ABB RobotStudio station: FinalProject_SP.rspag

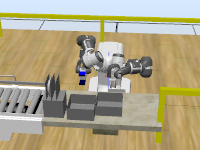
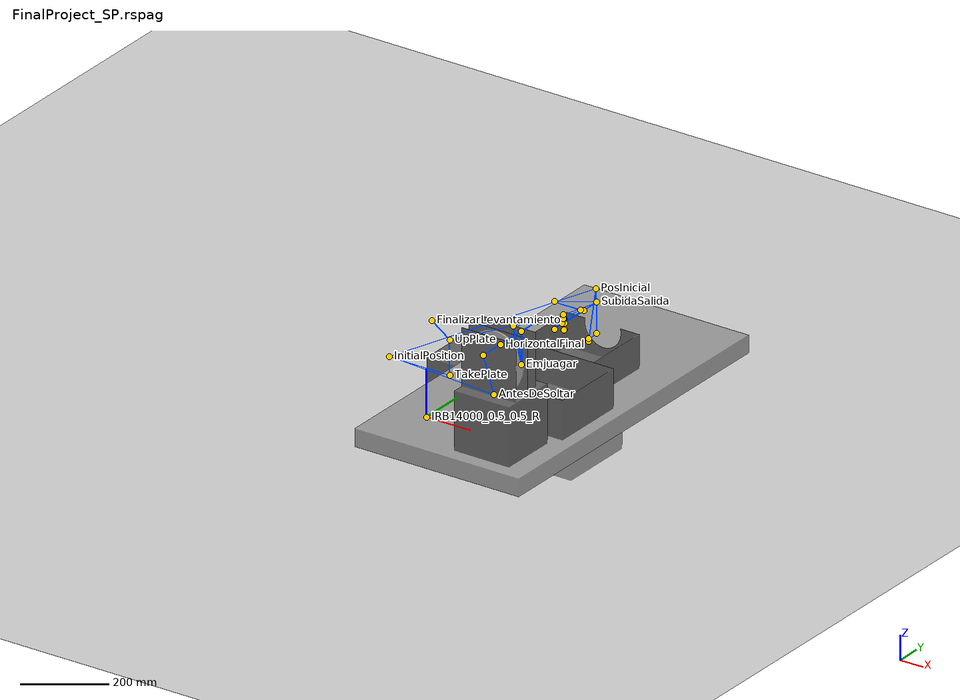
[picture v1: parts stored in the station drawn from their meshes, with robot base, taught points and paths (robot models come from the ABB library and are not in the file)]
--- station ---
Station FinalProject_SP (saved by RobotStudio 21.3.9648.0)
Controller IRB14000_1
  mechanical unit ROB_R: IRB14000_0.5_0.5_R, 6 joints, base frame (0, 0, 0) mm
  mechanical unit ROB_R_7: IRB14000_0.5_0.5_R, 1 joints, base frame (0, 0, 0) mm
  mechanical unit ROB_L: IRB14000_0.5_0.5_L, 6 joints, base frame (0, 0, 0) mm
  mechanical unit ROB_L_7: IRB14000_0.5_0.5_L, 1 joints, base frame (0, 0, 0) mm
Layout (positions relative to the parent item):
  - IRB14000_0.5_0.5 [mechanism, from Robots\IRB14000_0.5_0.5__01.rslib] at (0, 0, 0) mm
  - IRB14000_0.5_0.5_R [mechanism, from Robots\IRB14000_0.5_0.5__01.rslib] at (0, 0, 0) mm; joint values [-0.1923, -2.1323, -2.3764, 0.5232, 0.2776, 1.3361, 0.0448] (rad or m)
  - IRB14000_0.5_0.5_L [mechanism, from Robots\IRB14000_0.5_0.5__01.rslib] at (0, 0, 0) mm; joint values [2.2057, 0.7592, -2.9409, 0.6294, 1.2654, 1.781, -1.09] (rad or m)
  - LeftTool [mechanism] at (420.61, 55.54, 501.86) mm, rotated rx 176.45 ry 0.33 rz 178.52 deg; joint values [0, 0] (rad or m)
      TCP LeftTool_1 at (0, 0, 87) mm
      links: MainBody, R_Wash, L_Dry
  - floor [part] at (-1635.16, -1487.82, 4.97) mm, size 3000 x 3000 x 1 mm
  - Table [part] at (136.38, -477.32, 155.93) mm, size 450 x 900 x 45 mm
  - Plate [part] at (464.91, -410.88, 426.41) mm, rotated rx -91 ry -6 rz 0 deg, size 150 x 150 x 20 mm
  - SinkWsoap_3 [part] at (290.47, -67.3, 205.89) mm, size 200 x 200 x 85 mm
  - Sink_2 [part] at (461.13, -169.65, 206.31) mm, size 200 x 200 x 100 mm
  - Pieza_5 [part] at (260.22, -92.11, 0) mm, size 200 x 200 x 160 mm
  - RightGrip [mechanism] at (-31.94, -222.15, 256.56) mm, rotated rx -153.04 ry -89.35 rz -27.45 deg; joint values [0] (rad or m)
      TCP RightGrip at (0, 0, 85) mm
      links: Base, RightFinger, LeftFinger
  - 400_guide_2 [part, from Equipment\Conveyor Guide 400.rslib] at (524.45, -3451.19, -560.07) mm, rotated rx 0 ry 0 rz 89.33 deg
  - Pieza_8 [part] at (382.54, -381.93, 349.62) mm, size 159 x 2 x 150 mm
  - Pieza_9 [part] at (387.36, -418.51, 350.42) mm, size 150 x 1 x 150 mm
  - Pieza_10 [part] at (388.58, -447.06, 203.31) mm, size 150 x 150 x 150 mm
  - Pieza_11 [part], size 150 x 150 x 150 mm
  - Pieza_12 [part] at (388.74, -344.82, 350.01) mm, size 150 x 2 x 150 mm
  - Fence_2500_2 [graphiccomponentgroup, from Equipment\Fence_2500.rslib] at (-957.65, -1356.65, -1537.2) mm
    - Body 1 [part, from Equipment\Fence_2500.rslib]
    - Body 2 [part, from Equipment\Fence_2500.rslib]
  - Gate_2 [graphiccomponentgroup, from Equipment\Fence_Gate.rslib] at (-1379.63, -1420.32, -1615.31) mm, rotated rx 0 ry 0 rz -88.3 deg
    - Body 1 [part, from Equipment\Fence_Gate.rslib]
    - Body 2 [part, from Equipment\Fence_Gate.rslib]
    - Body 3 [part, from Equipment\Fence_Gate.rslib]
  - Gate_3 [graphiccomponentgroup, from Equipment\Fence_Gate.rslib] at (522.14, 1119.74, -1537.29) mm, rotated rx 0 ry 0 rz 90.8 deg
    - Body 1 [part, from Equipment\Fence_Gate.rslib]
    - Body 2 [part, from Equipment\Fence_Gate.rslib]
    - Body 3 [part, from Equipment\Fence_Gate.rslib]
  - Fence_740_2 [graphiccomponentgroup, from Equipment\Fence_740.rslib] at (506.71, 414.21, -1523.62) mm
    - Body 1 [part, from Equipment\Fence_740.rslib]
    - Body 2 [part, from Equipment\Fence_740.rslib]
Attachment: LeftTool is attached to IRB14000_0.5_0.5_L / Link7
Attachment: RightGrip is attached to IRB14000_0.5_0.5_R / Link7
EventTableEntry 3566: Group=, Trigger=DO_CloseGrip 3567, Actions=[EventTableActionMechanicalPose 3568, EventTableActionAttach 3576], Comment=, ActivationMode=2, Cyclic=false
EventTableTriggerIO 3567: IOValue=[1], IRC5Controller=? -1, Operator=0, SignalSource=IRB14000_1 1167
EventTableActionMechanicalPose 3568: VirtualSignal=SS_GripperClosed, Mechanism=RightGrip 3516, ToPoseName=Cerrado, VirtualSignalValue=[1]
EventTableEntry 3569: Group=, Trigger=DO_CloseGrip 3570, Actions=[EventTableActionMechanicalPose 5234, EventTableActionDetach 5235], Comment=, ActivationMode=2, Cyclic=false
EventTableTriggerIO 3570: IOValue=[0], IRC5Controller=? -1, Operator=0, SignalSource=IRB14000_1 1167
EventTableEntry 3572: Group=, Trigger=NOP 3573, Actions=[DI_GripperClosed 3575], Comment=, ActivationMode=2, Cyclic=false
EventTableTriggerLogic 3573: layoutX=8, layoutY=16, Operand1=SS_GripperClosed 3574, Operand2=? -1, Operator=4, Delay=1000
EventTableTriggerIO 3574: IOValue=[-1], IRC5Controller=? -1, Operator=0, SignalSource=FinalProject_SP 1
EventTableActionIO 3575: IOValue=[-1], IRC5Controller=? -1, SignalTarget=IRB14000_1 1167
EventTableActionAttach 3576: AttachmentParent=RightGrip 3516, AttachmentChild=Plate 3480, MountObject=false, Offset=[X=1, Y=0, Z=0, W=0, X=0, Y=1, Z=0, W=0, X=0, Y=0, Z=1, W=0, X=0, Y=0, Z=0, W=1], FlangeIndext=0, FindNearest=false
EventTableActionMechanicalPose 5234: VirtualSignal=SS_GripperClosed, Mechanism=RightGrip 3516, ToPoseName=Abierto, VirtualSignalValue=[0]
EventTableActionDetach 5235: AttachmentParent=RightGrip 3516, AttachmentChild=Plate 3480
EventTableTriggerIO 5306: IOValue=[1], IRC5Controller=? -1, Operator=0, SignalSource=IRB14000_1 1167
EventTableTriggerIO 5307: IOValue=[1], IRC5Controller=? -1, Operator=0, SignalSource=IRB14000_1 1167
EventTableTriggerIO 5308: IOValue=[0], IRC5Controller=? -1, Operator=0, SignalSource=IRB14000_1 1167
EventTableTriggerIO 5309: IOValue=[0], IRC5Controller=? -1, Operator=0, SignalSource=IRB14000_1 1167
EventTableTriggerLogic 5310: layoutX=8, layoutY=16, Operand1=SS_GripperClosed 3574, Operand2=? -1, Operator=4, Delay=1000
EventTableTriggerLogic 5311: layoutX=8, layoutY=16, Operand1=SS_GripperClosed 3574, Operand2=? -1, Operator=4, Delay=1000
Station signals: DI SS_GripperClosed
Targets, tools, work objects and paths stored in the station and not in the controller backup, written as RAPID:
! task T_ROB_R
MODULE Module1
  CONST robtarget SoltarObjeto:=[[612.086300085,-497.889224852,286.694545259],[0.048207182,0.789967534,-0.030176126,0.610505335],[1,1,1,4],[88.920010699,9E+09,9E+09,9E+09,9E+09,9E+09]];
ENDMODULE


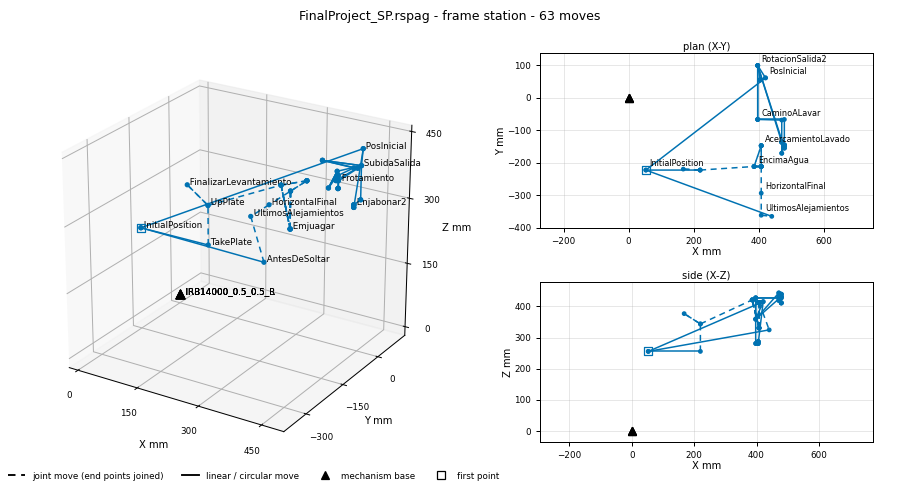
[picture p0: tool path of FinalProject_SP.rspag in frame station, 63 of 63 moves have a stored position in this frame; points joined in program order, loops and branches not executed]
--- Backups/IRB14000_1/RAPID/TASK1/PROGMOD/CalibData.mod ---
MODULE CalibData
    PERS tooldata RightGrip:=[TRUE,[[0,0,85],[1,0,0,0]],[0.32367,[0,0,17.36],[1,0,0,0],0,0,0]];
ENDMODULE

--- Backups/IRB14000_1/RAPID/TASK1/PROGMOD/Module1.mod ---
MODULE Module1
        CONST robtarget InitialPosition:=[[53.055314104,-222.870016919,255.704154577],[0.001177788,0.710631418,-0.004820161,0.703546989],[0,0,0,4],[-96.630018739,9E+09,9E+09,9E+09,9E+09,9E+09]];
    CONST robtarget TakePlate:=[[220.05553838,-222.870371261,255.704183843],[0.001177763,0.71063163,-0.004819912,0.703546777],[0,0,0,4],[-96.630024002,9E+09,9E+09,9E+09,9E+09,9E+09]];
    CONST robtarget UpPlate:=[[220.056150571,-222.871159309,343.704161267],[0.001177802,0.710632144,-0.004819416,0.703546262],[0,0,0,4],[-96.63002197,9E+09,9E+09,9E+09,9E+09,9E+09]];
    CONST robtarget FinalizarLevantamiento:=[[168.058261278,-219.873083697,376.704096677],[0.507683817,0.497248487,0.498428155,0.496558615],[0,1,-1,4],[-156.301628385,9E+09,9E+09,9E+09,9E+09,9E+09]];
    CONST robtarget Rotacion:=[[220.057272902,-222.872151334,343.70419509],[0.507684048,0.497248575,0.498427407,0.496559041],[0,0,-1,4],[-96.630018769,9E+09,9E+09,9E+09,9E+09,9E+09]];
    CONST robtarget EncimaAgua:=[[386.063679666,-211.876833518,420.702145472],[0.328812168,0.626355418,0.630919785,0.318593273],[0,2,-1,4],[98.779984801,9E+09,9E+09,9E+09,9E+09,9E+09]];
    CONST robtarget Emjuagar:=[[408.064481901,-211.877451805,330.701831056],[0.284000479,0.64705336,0.65232018,0.274124169],[0,2,-1,4],[102.139980128,9E+09,9E+09,9E+09,9E+09,9E+09]];
    CONST robtarget SalirDelAgua:=[[408.065294918,-211.877887738,412.70165188],[0.533074265,0.470579483,0.471179643,0.521897042],[-1,2,-1,4],[102.139982595,9E+09,9E+09,9E+09,9E+09,9E+09]];
    CONST robtarget AcomodoParaLavar:=[[408.065461711,-147.878021494,412.701612854],[0.53307426,0.470579475,0.471179771,0.521896939],[-1,2,-1,4],[102.139981571,9E+09,9E+09,9E+09,9E+09,9E+09]];
    CONST robtarget AcercamientoLavado:=[[408.066683421,-147.878727164,412.701031749],[0.533073873,0.470579276,0.471180857,0.521896533],[-1,2,-1,4],[102.139981352,9E+09,9E+09,9E+09,9E+09,9E+09]];
    CONST robtarget acercamiento2Lavado:=[[408.067566131,-147.879323271,412.700510834],[0.688610388,0.177278397,0.656761973,0.251101203],[0,2,-2,4],[122.539973578,9E+09,9E+09,9E+09,9E+09,9E+09]];
    CONST robtarget acercamiento2Lavado_2:=[[408.067566131,-147.879323271,412.700510834],[0.688610388,0.177278397,0.656761973,0.251101203],[0,2,-2,4],[122.539973578,9E+09,9E+09,9E+09,9E+09,9E+09]];
    CONST robtarget Emjuagar_2:=[[408.064481901,-211.877451805,330.701831056],[0.284000479,0.64705336,0.65232018,0.274124169],[0,2,-1,4],[102.139980128,9E+09,9E+09,9E+09,9E+09,9E+09]];
    CONST robtarget SalirDelAgua_2:=[[408.065294918,-211.877887738,412.70165188],[0.533074265,0.470579483,0.471179643,0.521897042],[-1,2,-1,4],[102.139982595,9E+09,9E+09,9E+09,9E+09,9E+09]];
    CONST robtarget Emjuagar_2_2:=[[408.064481901,-211.877451805,330.701831056],[0.284000479,0.64705336,0.65232018,0.274124169],[0,2,-1,4],[102.139980128,9E+09,9E+09,9E+09,9E+09,9E+09]];
    CONST robtarget SalirDelAgua_2_2:=[[408.065294918,-211.877887738,412.70165188],[0.533074265,0.470579483,0.471179643,0.521897042],[-1,2,-1,4],[102.139982595,9E+09,9E+09,9E+09,9E+09,9E+09]];
    CONST robtarget UltimoAlejamiento:=[[408.07197068,-293.881092513,412.699267968],[0.533045558,0.470580996,0.471214617,0.521893422],[-1,1,-1,4],[88.459990285,9E+09,9E+09,9E+09,9E+09,9E+09]];
    CONST robtarget HorizontalFinal:=[[408.072778957,-293.881627629,412.69925656],[0.044169035,0.709671302,-0.035834669,0.702233306],[-1,2,0,4],[80.980024532,9E+09,9E+09,9E+09,9E+09,9E+09]];
    CONST robtarget DejaElPlato:=[[408.076946424,-361.884549979,286.698372064],[0.044168859,0.709673429,-0.035831454,0.702231331],[-2,2,0,4],[94.167708654,9E+09,9E+09,9E+09,9E+09,9E+09]];
    CONST robtarget UltimosAlejamientos:=[[408.072401892,-361.881327349,412.699273877],[0.533045426,0.470580989,0.471214987,0.521893229],[-1,1,-1,4],[88.45998457,9E+09,9E+09,9E+09,9E+09,9E+09]];
    CONST robtarget AntesDeSoltar:=[[440.491875375,-365.351645888,324.606650036],[0.020610194,-0.811420808,-0.004875566,-0.584078523],[-1,1,0,4],[88.499974458,9E+09,9E+09,9E+09,9E+09,9E+09]];
!***********************************************************
    !***********************************************************
    PROC main()
        !Añada aquí su código
        MoveL InitialPosition,v500,fine,RightGrip\WObj:=wobj0;
        WaitDI DI_GripperClosed,0; !Gripper is opened
        MoveL TakePlate,v500,fine,RightGrip\WObj:=wobj0;
        SetDO DO_CloseGrip,1; !Close the gripper
        WaitDI DI_GripperClosed,1;!Gripper is closed
        MoveJ UpPlate,v500,z100,RightGrip\WObj:=wobj0;
        MoveJ FinalizarLevantamiento,v500,z100,RightGrip\WObj:=wobj0;
        MoveJ Rotacion,v500,z100,RightGrip\WObj:=wobj0;
        MoveJ EncimaAgua,v500,z100,RightGrip\WObj:=wobj0;
        MoveJ Emjuagar,v500,z100,RightGrip\WObj:=wobj0;
        MoveJ EncimaAgua,v500,z100,RightGrip\WObj:=wobj0;
        MoveJ Emjuagar,v500,z100,RightGrip\WObj:=wobj0;
        MoveJ SalirDelAgua,v500,fine,RightGrip\WObj:=wobj0;
        MoveJ Emjuagar_2,v500,z100,RightGrip\WObj:=wobj0;
        MoveJ SalirDelAgua_2,v500,fine,RightGrip\WObj:=wobj0;
        MoveJ Emjuagar_2_2,v500,z100,RightGrip\WObj:=wobj0;
        MoveJ SalirDelAgua_2_2,v500,fine,RightGrip\WObj:=wobj0;
        MoveJ AcercamientoLavado,v200,fine,RightGrip\WObj:=wobj0;
        MoveJ acercamiento2Lavado,v80,fine\Inpos:=stoptime1_5,RightGrip\WObj:=wobj0;
        MoveJ EncimaAgua,v500,fine,RightGrip\WObj:=wobj0;
        MoveJ Emjuagar,v500,fine,RightGrip\WObj:=wobj0;
        MoveJ EncimaAgua,v500,fine,RightGrip\WObj:=wobj0;
        MoveJ AcercamientoLavado,v500,fine,RightGrip\WObj:=wobj0;
        MoveJ acercamiento2Lavado,v500,fine\Inpos:=stoptime1_5,RightGrip\WObj:=wobj0;
        MoveJ AcercamientoLavado,v500,fine,RightGrip\WObj:=wobj0;
        MoveJ HorizontalFinal,v500,fine,RightGrip\WObj:=wobj0;
        MoveJ UltimosAlejamientos,v500,fine,RightGrip\WObj:=wobj0;
        MoveJ AntesDeSoltar,v1000,z100,RightGrip\WObj:=wobj0;
        WaitDI DI_GripperClosed,1; !Gripper is closed
        SetDO DO_CloseGrip,0; !Open the gripper
        WaitDI DI_GripperClosed,0;!Gripper is Open
        MoveL InitialPosition,v500,fine,RightGrip\WObj:=wobj0;

    ENDPROC
ENDMODULE

--- Backups/IRB14000_1/RAPID/TASK2/PROGMOD/CalibData.mod ---
MODULE CalibData
    PERS tooldata Dryer_Washer_1:=[TRUE,[[0,0,87],[1,0,0,0]],[0.306692,[0,-1.008,28.95],[1,0,0,0],0,0,0]];
    PERS tooldata Servo:=[TRUE,[[0,0,114.2],[1,0,0,0]],[0.229,[7.9,12.4,48.7],[1,0,0,0],0.00021,0.00023,0.00008]];
    PERS tooldata Camera:=[TRUE,[[-7.3,28.3,35.1],[0.5,-0.5,0.5,0.5]],[0.229,[7.9,12.4,48.7],[1,0,0,0],0.00021,0.00023,0.00008]];
    PERS tooldata LeftTool_1:=[TRUE,[[0,0,87],[1,0,0,0]],[0.30618,[0,-1.009,28.951],[1,0,0,0],0,0,0]];
ENDMODULE

--- Backups/IRB14000_1/RAPID/TASK2/PROGMOD/Module1.mod ---
MODULE Module1
        CONST robtarget PosInicial:=[[421.244619941,60.912152429,415.028508411],[0.003235703,0.012822081,0.999433724,0.030941171],[1,1,-1,0],[-178.213591377,9E+09,9E+09,9E+09,9E+09,9E+09]];
    CONST robtarget SegundaPos:=[[531.247516921,296.914105526,415.026910938],[0.003233398,0.012823194,0.999433674,0.030942565],[2,1,0,0],[-152.08998148,9E+09,9E+09,9E+09,9E+09,9E+09]];
    CONST robtarget AcomodoJabon:=[[531.249287785,296.915302981,283.026126749],[0.003677623,0.012703494,0.999904722,-0.003955191],[2,1,0,0],[-152.089982592,9E+09,9E+09,9E+09,9E+09,9E+09]];
    CONST robtarget SegundoAcomodo:=[[531.251888568,200.917989137,287.024191767],[0.003743422,-0.004748162,0.999974161,-0.003888287],[2,1,0,0],[-151.229980314,9E+09,9E+09,9E+09,9E+09,9E+09]];
    CONST robtarget Encaje:=[[531.253237835,180.919326703,287.022987741],[0.000816881,0.005991691,-0.69184437,0.722021329],[1,0,0,0],[-151.230030681,9E+09,9E+09,9E+09,9E+09,9E+09]];
    CONST robtarget Lavar:=[[531.256510861,180.923529425,243.019596759],[0.691724056,0.721807274,0.012895058,-0.018595875],[1,0,2,0],[-151.230032118,9E+09,9E+09,9E+09,9E+09,9E+09]];
    CONST robtarget BajaASoap:=[[421.245417577,58.912937477,271.02790989],[0.003234896,0.012822498,0.999433703,0.030941751],[1,1,-1,0],[-168.160186005,9E+09,9E+09,9E+09,9E+09,9E+09]];
    CONST robtarget Enjabonar:=[[405.248437711,54.917136531,281.025032798],[0.704216771,0.709627455,0.013003664,-0.018398897],[1,0,-1,0],[-152.810020426,9E+09,9E+09,9E+09,9E+09,9E+09]];
    CONST robtarget Enjabonar2:=[[405.249506318,54.918706238,287.024012367],[0.704215896,0.709628284,0.01300405,-0.018400126],[1,0,-1,0],[-152.810017528,9E+09,9E+09,9E+09,9E+09,9E+09]];
    CONST robtarget RotacionSalida:=[[405.250228712,54.919564027,287.023505096],[0.221162905,0.974976545,0.020779228,-0.00871373],[2,1,-3,0],[-151.089999947,9E+09,9E+09,9E+09,9E+09,9E+09]];
    CONST robtarget RotacionSalida2:=[[397.251225339,98.920933427,281.022531986],[0.221162073,0.974976732,0.02077867,-0.008715334],[2,1,-2,0],[-144.406554524,9E+09,9E+09,9E+09,9E+09,9E+09]];
    CONST robtarget SalidaRotacion:=[[397.257647968,98.928500253,325.017724075],[0.047711709,0.997734001,0.026081142,-0.039626132],[2,1,-3,0],[-141.807190023,9E+09,9E+09,9E+09,9E+09,9E+09]];
    CONST robtarget AfueraRotacion:=[[397.252338551,98.922405636,281.021643738],[0.704213985,0.709630106,0.01300311,-0.018403658],[2,0,-1,0],[-143.450011398,9E+09,9E+09,9E+09,9E+09,9E+09]];
    CONST robtarget SubidaSalida:=[[397.253299337,98.923503411,359.020949108],[0.704213348,0.709630696,0.01300383,-0.018404812],[2,0,-1,0],[-137.099990443,9E+09,9E+09,9E+09,9E+09,9E+09]];
    CONST robtarget CaminoALavar:=[[397.254740388,-67.075582852,427.02014683],[0.704212985,0.709631027,0.013003711,-0.018405994],[2,-1,-1,0],[-138.173949069,9E+09,9E+09,9E+09,9E+09,9E+09]];
    CONST robtarget AcercamientoLavado:=[[397.255236135,-67.075179426,427.019791885],[0.465965923,0.88451561,0.017817153,-0.013800111],[2,0,-3,0],[-162.169977355,9E+09,9E+09,9E+09,9E+09,9E+09]];
    CONST robtarget Acercamiento2:=[[479.255350173,-67.075059648,427.019646749],[0.465965804,0.884515669,0.017817213,-0.013800279],[1,0,-2,0],[-162.169971229,9E+09,9E+09,9E+09,9E+09,9E+09]];
    CONST robtarget Frotamiento:=[[479.256631089,-145.074003616,427.018181948],[0.465964987,0.884516076,0.01781704,-0.013802011],[1,0,-3,0],[-162.170033234,9E+09,9E+09,9E+09,9E+09,9E+09]];
    CONST robtarget Bajo1:=[[479.257332601,-145.073375587,411.017323942],[0.465964389,0.88451639,0.017816677,-0.013802499],[1,0,-3,0],[-161.630016937,9E+09,9E+09,9E+09,9E+09,9E+09]];
    CONST robtarget Bajo2:=[[479.257619446,-147.073077759,411.016894097],[0.465964074,0.88451655,0.017816607,-0.013802987],[1,0,-3,0],[-161.630015461,9E+09,9E+09,9E+09,9E+09,9E+09]];
    CONST robtarget RotacionPenultima:=[[479.257920024,-147.072880521,411.016622834],[0.826677125,0.562225014,0.009251006,-0.020551967],[1,-1,-1,0],[-161.339982134,9E+09,9E+09,9E+09,9E+09,9E+09]];
    CONST robtarget CambioDeLado:=[[479.258634617,-147.072192495,411.01554837],[0.00925188,0.020552151,-0.826677374,0.562224626],[1,0,0,0],[-161.339985535,9E+09,9E+09,9E+09,9E+09,9E+09]];
    CONST robtarget Frotamiento2:=[[479.26034828,-147.070681628,439.013141409],[0.009254109,0.020552461,-0.826678168,0.562223411],[1,0,0,0],[-161.339982258,9E+09,9E+09,9E+09,9E+09,9E+09]];
    CONST robtarget BajadaLimpia:=[[479.261993602,-155.069467218,431.011459943],[0.009256027,0.020552551,-0.826678574,0.56222278],[1,0,0,0],[-161.340012683,9E+09,9E+09,9E+09,9E+09,9E+09]];
    CONST robtarget CaminoALavar_2:=[[397.254740388,-67.075582852,427.02014683],[0.704212985,0.709631027,0.013003711,-0.018405994],[2,-1,-1,0],[-138.173949069,9E+09,9E+09,9E+09,9E+09,9E+09]];
    CONST robtarget AcercamientoLavado_2:=[[397.255236135,-67.075179426,427.019791885],[0.465965923,0.88451561,0.017817153,-0.013800111],[2,0,-3,0],[-162.169977355,9E+09,9E+09,9E+09,9E+09,9E+09]];
    CONST robtarget Acercamiento2_2:=[[479.255350173,-67.075059648,427.019646749],[0.465965804,0.884515669,0.017817213,-0.013800279],[1,0,-2,0],[-162.169971229,9E+09,9E+09,9E+09,9E+09,9E+09]];
    CONST robtarget Frotamiento_2:=[[479.256631089,-145.074003616,427.018181948],[0.465964987,0.884516076,0.01781704,-0.013802011],[1,0,-3,0],[-162.170033234,9E+09,9E+09,9E+09,9E+09,9E+09]];
    CONST robtarget Bajo1_2:=[[479.257332601,-145.073375587,411.017323942],[0.465964389,0.88451639,0.017816677,-0.013802499],[1,0,-3,0],[-161.630016937,9E+09,9E+09,9E+09,9E+09,9E+09]];
    CONST robtarget Bajo2_2:=[[479.257619446,-147.073077759,411.016894097],[0.465964074,0.88451655,0.017816607,-0.013802987],[1,0,-3,0],[-161.630015461,9E+09,9E+09,9E+09,9E+09,9E+09]];
    CONST robtarget RotacionPenultima_2:=[[479.257920024,-147.072880521,411.016622834],[0.826677125,0.562225014,0.009251006,-0.020551967],[1,-1,-1,0],[-161.339982134,9E+09,9E+09,9E+09,9E+09,9E+09]];
    CONST robtarget Frotamiento2_2:=[[479.26034828,-147.070681628,439.013141409],[0.009254109,0.020552461,-0.826678168,0.562223411],[1,0,0,0],[-161.339982258,9E+09,9E+09,9E+09,9E+09,9E+09]];
    CONST robtarget BajadaLimpia_3:=[[479.261993602,-155.069467218,431.011459943],[0.009256027,0.020552551,-0.826678574,0.56222278],[1,0,0,0],[-161.340012683,9E+09,9E+09,9E+09,9E+09,9E+09]];
    CONST robtarget BajadaLimpia_2:=[[479.261993602,-155.069467218,431.011459943],[0.009256027,0.020552551,-0.826678574,0.56222278],[1,0,0,0],[-161.340012683,9E+09,9E+09,9E+09,9E+09,9E+09]];
    CONST robtarget Frotamiento2_3:=[[479.26034828,-147.070681628,439.013141409],[0.009254109,0.020552461,-0.826678168,0.562223411],[1,0,0,0],[-161.339982258,9E+09,9E+09,9E+09,9E+09,9E+09]];
    CONST robtarget UltimaAproximacion:=[[471.256137044,-69.074277916,427.018433556],[0.465965108,0.884516007,0.017817773,-0.013801412],[1,0,-2,0],[-161.699970308,9E+09,9E+09,9E+09,9E+09,9E+09]];
    CONST robtarget UltimoToque:=[[471.257048398,-137.073488671,433.016805154],[0.46596401,0.884516566,0.017817963,-0.013802425],[1,0,-3,0],[-161.69997174,9E+09,9E+09,9E+09,9E+09,9E+09]];
    CONST robtarget UtimaInclinacion:=[[471.258027829,-137.072698082,433.015349989],[0.570285555,0.821137245,0.01600292,-0.01587192],[1,0,-2,0],[-161.229978292,9E+09,9E+09,9E+09,9E+09,9E+09]];
    CONST robtarget FrotamientoFinal:=[[471.261017466,-171.069905885,419.010772839],[0.570283267,0.821138759,0.016003358,-0.015875366],[1,0,-2,0],[-161.229980195,9E+09,9E+09,9E+09,9E+09,9E+09]];
    CONST robtarget FrotacionFinal:=[[471.264656463,-137.066480694,443.005226558],[0.570280059,0.821140864,0.016004384,-0.015880669],[1,0,-2,0],[-161.22997221,9E+09,9E+09,9E+09,9E+09,9E+09]];
    CONST robtarget FrotamientoFinal_2:=[[471.261017466,-171.069905885,419.010772839],[0.570283267,0.821138759,0.016003358,-0.015875366],[1,0,-2,0],[-161.229980195,9E+09,9E+09,9E+09,9E+09,9E+09]];
    CONST robtarget FrotacionFinal_2:=[[471.264656463,-137.066480694,443.005226558],[0.570280059,0.821140864,0.016004384,-0.015880669],[1,0,-2,0],[-161.22997221,9E+09,9E+09,9E+09,9E+09,9E+09]];
    CONST robtarget SubidaSalida_2:=[[397.253299337,98.923503411,359.020949108],[0.704213348,0.709630696,0.01300383,-0.018404812],[2,0,-1,0],[-137.099990443,9E+09,9E+09,9E+09,9E+09,9E+09]];
!***********************************************************
    !
    ! Módulo:  Module1
    !
    ! Descripción:
    !   <Introduzca la descripción aquí>
    !
    ! Autor: sr118
    !
    ! Versión: 1.0
    !
    !***********************************************************


    !***********************************************************
    !
    ! Procedimiento Main
    !
    !   Este es el punto de entrada de su programa
    !
    !***********************************************************
    PROC main()
        !Añada aquí su código
        MoveL PosInicial,v500,fine,LeftTool_1\WObj:=wobj0;
        MoveL Enjabonar,v500,fine,LeftTool_1\WObj:=wobj0;
        MoveL Enjabonar2,v500,fine,LeftTool_1\WObj:=wobj0;
        MoveL Enjabonar,v500,fine,LeftTool_1\WObj:=wobj0;
        MoveL Enjabonar2,v500,fine,LeftTool_1\WObj:=wobj0;
        MoveL Enjabonar,v500,fine,LeftTool_1\WObj:=wobj0;
        MoveL Enjabonar2,v500,z100,LeftTool_1\WObj:=wobj0;
        MoveL RotacionSalida,v500,fine,LeftTool_1\WObj:=wobj0;
        MoveL RotacionSalida2,v500,fine,LeftTool_1\WObj:=wobj0;
        MoveL AfueraRotacion,v500,fine,LeftTool_1\WObj:=wobj0;
        MoveL SubidaSalida,v500,fine,LeftTool_1\WObj:=wobj0;
        MoveL CaminoALavar,v500,fine,LeftTool_1\WObj:=wobj0;
        MoveL AcercamientoLavado,v500,fine,LeftTool_1\WObj:=wobj0;
        MoveL Acercamiento2,v500,fine,LeftTool_1\WObj:=wobj0;
        MoveL Frotamiento,v500,z100,LeftTool_1\WObj:=wobj0;
        MoveL Bajo1,v500,fine,LeftTool_1\WObj:=wobj0;
        MoveL Bajo2,v500,fine,LeftTool_1\WObj:=wobj0;
        MoveL RotacionPenultima,v500,fine,LeftTool_1\WObj:=wobj0;
        MoveL CambioDeLado,v500,fine,LeftTool_1\WObj:=wobj0;
        MoveL Frotamiento2,v500,fine,LeftTool_1\WObj:=wobj0;
        MoveL BajadaLimpia,v500,z100,LeftTool_1\WObj:=wobj0;
        MoveL Frotamiento2,v500,fine,LeftTool_1\WObj:=wobj0;
        MoveL BajadaLimpia,v500,fine,LeftTool_1\WObj:=wobj0;
        MoveL Frotamiento2,v500,fine,LeftTool_1\WObj:=wobj0;
        MoveL BajadaLimpia,v500,fine,LeftTool_1\WObj:=wobj0;
        MoveL SubidaSalida,v500,fine,LeftTool_1\WObj:=wobj0;
        MoveL CaminoALavar_2,v500,fine,LeftTool_1\WObj:=wobj0;
        MoveL AcercamientoLavado_2,v500,fine,LeftTool_1\WObj:=wobj0;
        MoveL UltimaAproximacion,v500,fine,LeftTool_1\WObj:=wobj0;
        MoveL UltimoToque,v500,fine,LeftTool_1\WObj:=wobj0;
        MoveL UtimaInclinacion,v500,fine,LeftTool_1\WObj:=wobj0;
        MoveL FrotamientoFinal,v500,fine,LeftTool_1\WObj:=wobj0;
        MoveL FrotacionFinal,v500,fine,LeftTool_1\WObj:=wobj0;
        MoveL FrotamientoFinal_2,v500,fine,LeftTool_1\WObj:=wobj0;
        MoveL FrotacionFinal_2,v500,fine,LeftTool_1\WObj:=wobj0;
        MoveL SubidaSalida_2,v500,fine,LeftTool_1\WObj:=wobj0;
        MoveL PosInicial,v500,fine,LeftTool_1\WObj:=wobj0;
    ENDPROC
ENDMODULE

--- Backups/IRB14000_1/SYSPAR/EIO.cfg ---
EIO:CFG_1.0:6:1::
#
SYSSIG_IN:

      -Signal "Collision_Avoidance" -Action "CollAvoidance"
#
INDUSTRIAL_NETWORK:

      -Name "EtherNetIP" -Connection "Private Network"\
      -Label "EtherNet/IP Adapter Network"

      -Name "DeviceNet" -Label "DeviceNet Master/Slave Network" -Address "2"
#
EIO_CROSS:

      -Name "Cross_Signal_Lamp" -Res "Signal_Lamp" -Act1 "DRV1BRAKE"
#
EIO_SIGNAL_SAFELEVEL:

      -Name "FlangePowerSafeLevel" -ActionWhenStartup "Last"
#
DEVICENET_DEVICE:

      -Name "D652_10" -VendorName "ABB Robotics" -ProductName "24 VDC Unit"\
      -Address 10 -ProductCode 26 -DeviceType 7 -ConnectionType "COS"\
      -OutputSize 2 -InputSize 2
#
DEVICENET_INTERNAL_DEVICE:

      -Name "DN_Internal_Device" -VendorName "ABB Robotics"\
      -ProductName "DeviceNet Internal Slave Device"
#
ETHERNETIP_INTERNAL_DEVICE:

      -Name "EN_Internal_Device" -VendorName "ABB Robotics"\
      -ProductName "EtherNet/IP Internal Adapter Device"
#
EIO_SIGNAL:

      -Name "custom_DI_0" -SignalType "DI" -Device "D652_10" -DeviceMap "0"

      -Name "custom_DI_1" -SignalType "DI" -Device "D652_10" -DeviceMap "1"

      -Name "custom_DI_2" -SignalType "DI" -Device "D652_10" -DeviceMap "2"

      -Name "custom_DI_3" -SignalType "DI" -Device "D652_10" -DeviceMap "3"

      -Name "custom_DI_4" -SignalType "DI" -Device "D652_10" -DeviceMap "4"

      -Name "custom_DI_5" -SignalType "DI" -Device "D652_10" -DeviceMap "5"

      -Name "custom_DI_6" -SignalType "DI" -Device "D652_10" -DeviceMap "6"

      -Name "custom_DI_7" -SignalType "DI" -Device "D652_10" -DeviceMap "7"

      -Name "custom_DO_0" -SignalType "DO" -Device "D652_10" -DeviceMap "0"

      -Name "custom_DO_1" -SignalType "DO" -Device "D652_10" -DeviceMap "1"

      -Name "custom_DO_2" -SignalType "DO" -Device "D652_10" -DeviceMap "2"

      -Name "custom_DO_3" -SignalType "DO" -Device "D652_10" -DeviceMap "3"

      -Name "custom_DO_4" -SignalType "DO" -Device "D652_10" -DeviceMap "4"

      -Name "custom_DO_5" -SignalType "DO" -Device "D652_10" -DeviceMap "5"

      -Name "custom_DO_6" -SignalType "DO" -Device "D652_10" -DeviceMap "6"

      -Name "custom_DO_7" -SignalType "DO" -Device "D652_10" -DeviceMap "7"

      -Name "hall_sensor_joint_1" -SignalType "DI" -Device "D652_10"\
      -DeviceMap "8"

      -Name "hall_sensor_joint_2" -SignalType "DI" -Device "D652_10"\
      -DeviceMap "9"

      -Name "hall_sensor_joint_3" -SignalType "DI" -Device "D652_10"\
      -DeviceMap "11"

      -Name "hall_sensor_joint_4" -SignalType "DI" -Device "D652_10"\
      -DeviceMap "12"

      -Name "hall_sensor_joint_5" -SignalType "DI" -Device "D652_10"\
      -DeviceMap "13"

      -Name "hall_sensor_joint_6" -SignalType "DI" -Device "D652_10"\
      -DeviceMap "14"

      -Name "hall_sensor_joint_7" -SignalType "DI" -Device "D652_10"\
      -DeviceMap "10"

      -Name "hall_sensor_24V_ROB_R" -SignalType "DO" -Device "D652_10"\
      -DeviceMap "8"

      -Name "hall_sensor_24V_ROB_L" -SignalType "DO" -Device "D652_10"\
      -DeviceMap "9"

      -Name "flange_24V_ROB_R" -SignalType "DO" -Device "D652_10"\
      -DeviceMap "10" -SafeLevel "FlangePowerSafeLevel"

      -Name "flange_24V_ROB_L" -SignalType "DO" -Device "D652_10"\
      -DeviceMap "11" -SafeLevel "FlangePowerSafeLevel"

      -Name "Signal_Lamp" -SignalType "DO" -Device "D652_10" -DeviceMap "12"

      -Name "Collision_Avoidance" -SignalType "DO" -Access "All" -Default 1

      -Name "DO_CloseGrip" -SignalType "DO" -Access "All"

      -Name "DI_GripperClosed" -SignalType "DI" -Access "All"
